FUNCTION_BLOCK CLIENT_0_1 (* Single-RD Client Interface *)
  (* Standard: 61499-1; Function: Communication; Description: 0SD/1RD Client *)
  (* Version 0.0, 2001-09-18, JHC, Rockwell Automation *)
  (* Compiler header: package fb.rt.net; *)
  (* Compiler Java IBM VisualAge 3.0 *)
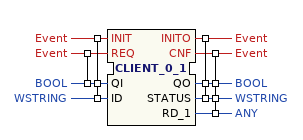
  EVENT_INPUT
    INIT WITH QI, ID; (* Service Initialization *)
    REQ WITH QI; (* Service Request *)
  END_EVENT
  EVENT_OUTPUT
    INITO WITH QO, STATUS; (* Initialization Confirm *)
    CNF WITH QO, STATUS, RD_1; (* Service Confirmation *)
  END_EVENT
  VAR_INPUT
    QI : BOOL; (* Event Input Qualifier *)
    ID : WSTRING; (* Connection Identifier *)
  END_VAR
  VAR_OUTPUT
    QO : BOOL; (* Event Output Qualifier *)
    STATUS : WSTRING; (* Service Status *)
    RD_1 : ANY; (* Received Data *)
  END_VAR
END_FUNCTION_BLOCK
